(*
DESCRIPTION: This function block parses a the part "flags" of the diagnostic message according to the
             ETG.1020 protocol enhancements.
*)
FUNCTION_BLOCK FB_DiagnosticMessageFlagsParser
VAR_INPUT
    anFlagsBuffer : ARRAY[1..2] OF BYTE;
END_VAR
VAR_OUTPUT
    stFlags : ST_FLAGS;
END_VAR
VAR
    nFlags : BYTE;
END_VAR

nFlags.0 := anFlagsBuffer[1].0;
nFlags.1 := anFlagsBuffer[1].1;
nFlags.2 := anFlagsBuffer[1].2;
nFlags.3 := anFlagsBuffer[1].3;

{analysis -34}
//IF nFlags >= 10#0 AND nFlags <= 10#2 THEN
IF nFlags >= 10#1 AND nFlags <= 10#2 THEN
    stFlags.eDiagnosisType := nFlags;
ELSE
    stFlags.eDiagnosisType := E_DIAGNOSISTYPE.Unspecified;
END_IF
{analysis +34}

IF anFlagsBuffer[1].4 THEN
    stFlags.eTimeStampType := E_TIMESTAMPTYPE.Local;
ELSE
    stFlags.eTimeStampType := E_TIMESTAMPTYPE.Global;
END_IF

stFlags.nNumberOfParametersInDiagnosisMessage := BYTE_TO_USINT(anFlagsBuffer[2]);

END_FUNCTION_BLOCK

(* stored: Version 1.1.0.1, ProductVersion 3.1.4022.12
   POU FB_DiagnosticMessageFlagsParser: Id {958e46be-3e7d-422e-a657-01a3d5ad4365}, SpecialFunc None *)
